// TIA Portal V16 export
// export: Created 2022-09-01T13:37:26.1417235Z, ExportSetting WithDefaults, DisplayName Totally Integrated Automation Portal, DisplayVersion V16, DisplayName TIA Portal Version Control Interface, DisplayVersion V16, DisplayName TIA Portal Openness, DisplayVersion V16, DisplayName STEP 7 Professional, DisplayVersion V16, DisplayName STEP 7 Safety, DisplayVersion V16, DisplayName WinCC Advanced, DisplayVersion V16
VAR_GLOBAL   // PLC tag table "Níveis"
   LSH001_TK00 AT %I0.6 : Bool;
   LSL001_TK00 AT %I1.0 : Bool;
   LSH501_TK05 AT %I1.3 : Bool;
   LSL501_TK05 AT %I1.4 : Bool;
   LSH101_TK01 AT %I1.1 : Bool;
   LS201_TK02 AT %IW12 : Word;
   LS301_TK03 AT %IW14 : Word;
   LSL101_TK01 AT %I1.2 : Bool;
   LSM001_TK00 AT %I0.7 : Bool;
END_VAR
